Staubli VAL3: loadPage.pgx

program loadPage(string x_sPage, string& x_sItems[])
// load the next page
  local num i
  local string l_sMessage
begin
end
